(* CODESYS project plc_207_climat.project

Project tree, tasks and I/O mapping:
  Device : Owen SPK2xx 03.CS.WEB, Owen, order no. 023, version 3.5.4.20
    application Application
      libraries: Standard, * (System); VisuDialogs, * (System)
      task MainTask (cyclic, interval t#10ms, priority 1) calls PLC_PRG
      task VISU_TASK (cyclic, interval 100 ms, priority 31) calls VisuElems.Visu_Prg
      task AlarmManagerTask (cyclic, interval 50 ms, priority 31) calls AlarmManager.Alarm_Prg
      task Taskbus (cyclic, interval t#200ms, priority 1) calls MV110_16DN, MV110_8A, MU110_8P
      program PLC_PRG [ST]
      visualisation log_visu
      function two_word_to_real [ST]
      image pool ImagePool
      Alarm Configuration
        text list AlarmGroup
        alarm group AlarmGroup
            11 [Info]: Comparison Equal, ExpressionToCompare FALSE, Expression PLC_PRG.heating_on_level_1 - "Обогрев выключен, уровень 1"
            14 [Info]: Comparison Equal, ExpressionToCompare FALSE, Expression PLC_PRG.fire_alarm - "Пожара нет"
            8 [Info]: Comparison Equal, ExpressionToCompare FALSE, Expression PLC_PRG.air_valves_open - "Заслонки закрыты"
            9 [Info]: Comparison Equal, ExpressionToCompare FALSE, Expression PLC_PRG.fan_on_1 - "Вентилятор 1 выключен"
            12 [Info]: Comparison Equal, ExpressionToCompare FALSE, Expression PLC_PRG.heating_on_level_2 - "Обогрев выключен, уровень 2"
            0 [Error]: Comparison Equal, ExpressionToCompare TRUE, Expression PLC_PRG.air_valves_open - "Заслонки открыты"
            1 [Error]: Comparison Equal, ExpressionToCompare TRUE, Expression PLC_PRG.fan_on_1 - "Вентилятор 1 включен"
            2 [Error]: Comparison Equal, ExpressionToCompare TRUE, Expression PLC_PRG.fan_on_2 - "Вентилятор 2 включен"
            15 [Info]: Comparison Equal, ExpressionToCompare FALSE, Expression PLC_PRG.extinction_voltage - "Наличие напряжения на СШ"
            4 [Error]: Comparison Equal, ExpressionToCompare TRUE, Expression PLC_PRG.heating_on_level_2 - "Обогрев включен, уровень 2"
            5 [Error]: Comparison Equal, ExpressionToCompare TRUE, Expression PLC_PRG.automation_off - "Автоматика выключена"
            6 [Error]: Comparison Equal, ExpressionToCompare TRUE, Expression PLC_PRG.fire_alarm - "Пожар"
            7 [Error]: Comparison Equal, ExpressionToCompare TRUE, Expression PLC_PRG.extinction_voltage - "Исчезновение напряжения на СШ"
            13 [Info]: Comparison Equal, ExpressionToCompare TRUE, Expression PLC_PRG.automation_on - "Автоматика включена"
            3 [Error]: Comparison Equal, ExpressionToCompare TRUE, Expression PLC_PRG.heating_on_level_1 - "Обогрев включен, уровень 1"
            10 [Info]: Comparison Equal, ExpressionToCompare FALSE, Expression PLC_PRG.fan_on_2 - "Вентилятор 2 выключен"
        AlarmStorage
        alarm class Info (priority 10, acknowledge REP)
        alarm class Error (priority 20, acknowledge REP)
      visualisation log_visu_history
      function block BLINK [ST]
      visualisation main
      data type MAIN_STATE
    Modbus : Modbus COM, 3S - Smart Software Solutions GmbH, version 3.4.0.0
        settings: DataBits = 8; StopBits = 1; ComPort = 3
      Modbus_Master : Modbus Master, COM Port, 3S - Smart Software Solutions GmbH, version 3.5.4.0
          settings: Transmission = 'RTU'; ResponseTimeout = 300; TimeBetweenFrames = 50
        MV110_16DN : Modbus Slave, COM Port, 3S - Smart Software Solutions GmbH, version 3.5.4.0
            settings: SlaveAddress = 1; ResponseTimeout = 200; UseExtendedFunctionCodes = TRUE; Channel0.Function Code = 3; Channel0.Read Offset = 16#0033; Channel0.Read Length = 1; Channel0.Write Offset = 0; Channel0.Write Length = 0; Channel0.Cycle Time = 100
            input  Application.PLC_PRG.fan_on_1 : BOOL  // Channel0.Channel0.Bit0
            input  Application.PLC_PRG.fan_on_2 : BOOL  // Channel0.Channel0.Bit1
            input  Application.PLC_PRG.heating_on_level_1 : BOOL  // Channel0.Channel0.Bit2
            input  Application.PLC_PRG.heating_on_level_2 : BOOL  // Channel0.Channel0.Bit3
            input  Application.PLC_PRG.air_valves_open : BOOL  // Channel0.Channel0.Bit4
            input  Application.PLC_PRG.automation_off : BOOL  // Channel0.Channel0.Bit6
            input  Application.PLC_PRG.fire_alarm : BOOL  // Channel0.Channel0.Bit7
            input  Application.PLC_PRG.extinction_voltage_r : BOOL  // Channel0.Channel0.Bit8
            unmapped channels: Channel0
        MU110_8P : Modbus Slave, COM Port, 3S - Smart Software Solutions GmbH, version 3.5.4.0
            settings: SlaveAddress = 2; ResponseTimeout = 200; UseExtendedFunctionCodes = TRUE; Channel0.Function Code = 15; Channel0.Read Offset = 0; Channel0.Read Length = 0; Channel0.Write Offset = 16#0000; Channel0.Write Length = 8; Channel0.Cycle Time = 100
            output Application.PLC_PRG.ctr_vent : BOOL  // Channel0.Channel0.Bit0
            output Application.PLC_PRG.ctr_heating_level_1 : BOOL  // Channel0.Channel0.Bit1
            output Application.PLC_PRG.ctr_heating_level_2 : BOOL  // Channel0.Channel0.Bit2
            output Application.PLC_PRG.ctr_air_valves_open : BOOL  // Channel0.Channel0.Bit3
            output Application.PLC_PRG.ctr_low_temp_alarm : BOOL  // Channel0.Channel0.Bit4
            output Application.PLC_PRG.ctr_high_temp_alarm : BOOL  // Channel0.Channel0.Bit5
            output Application.PLC_PRG.ctr_fire_alarm : BOOL  // Channel0.Channel0.Bit6
            output Application.PLC_PRG.ctr_no_voltage_alarm : BOOL  // Channel0.Channel0.Bit7
            unmapped channels: Channel0
        MV110_8A : Modbus Slave, COM Port, 3S - Smart Software Solutions GmbH, version 3.5.4.0
            settings: SlaveAddress = 3; ResponseTimeout = 200; UseExtendedFunctionCodes = TRUE; Channel0.Function Code = 3; Channel0.Read Offset = 16#0004; Channel0.Read Length = 26; Channel0.Write Offset = 0; Channel0.Write Length = 0; Channel0.Cycle Time = 100
            input  Application.PLC_PRG.arr_t_outside[0] : WORD  // Channel0.Channel0
            input  Application.PLC_PRG.arr_t_outside[1] : WORD  // Channel0.Channel0
            input  Application.PLC_PRG.arr_t_inside_1[0] : WORD  // Channel0.Channel0
            input  Application.PLC_PRG.arr_t_inside_1[1] : WORD  // Channel0.Channel0
            input  Application.PLC_PRG.arr_t_inside_2[0] : WORD  // Channel0.Channel0
            input  Application.PLC_PRG.arr_t_inside_2[1] : WORD  // Channel0.Channel0
            unmapped channels: Channel0
    Modbus_OUT : Modbus COM, 3S - Smart Software Solutions GmbH, version 3.4.0.0
        settings: DataBits = 8; StopBits = 1; ComPort = 4
      Modbus_Slave : Modbus Serial Device, 3S - Smart Software Solutions GmbH, version 3.5.3.80
          settings: Unit-ID = 3
          output Application.PLC_PRG.fan_on_1 : BOOL  // Outputs.Outputs.Bit0
          output Application.PLC_PRG.fan_on_2 : BOOL  // Outputs.Outputs.Bit1
          output Application.PLC_PRG.heating_on_level_1 : BOOL  // Outputs.Outputs.Bit2
          output Application.PLC_PRG.heating_on_level_2 : BOOL  // Outputs.Outputs.Bit3
          output Application.PLC_PRG.air_valves_open : BOOL  // Outputs.Outputs.Bit4
          output Application.PLC_PRG.automation_off : BOOL  // Outputs.Outputs.Bit5
          output Application.PLC_PRG.fire_alarm : BOOL  // Outputs.Outputs.Bit6
          output Application.PLC_PRG.extinction_voltage_r : BOOL  // Outputs.Outputs.Bit7
          output Application.PLC_PRG.ctr_low_temp_alarm : BOOL  // Outputs.Outputs.Bit8
          output Application.PLC_PRG.ctr_high_temp_alarm : BOOL  // Outputs.Outputs.Bit9
          output Application.PLC_PRG.arr_t_outside[0] : WORD  // Outputs.Outputs
          output Application.PLC_PRG.arr_t_outside[1] : WORD  // Outputs.Outputs
          output Application.PLC_PRG.arr_t_inside_1[0] : WORD  // Outputs.Outputs
          output Application.PLC_PRG.arr_t_inside_1[1] : WORD  // Outputs.Outputs
          output Application.PLC_PRG.arr_t_inside_2[0] : WORD  // Outputs.Outputs
          output Application.PLC_PRG.arr_t_inside_2[1] : WORD  // Outputs.Outputs
          unmapped channels: Inputs, Outputs
  text list GlobalTextList
  5ce3da45-db07-42e7-a21c-a00fff4ed8f6|D:\по щсу\ДЭС\visu\zit.jpg
  5ce3da45-db07-42e7-a21c-a00fff4ed8f6|D:\по щсу\ДЭС\visu\entel.jpg
  5ce3da45-db07-42e7-a21c-a00fff4ed8f6|C:\Users\Maxim\Desktop\mie110-3m.jpg
  5ce3da45-db07-42e7-a21c-a00fff4ed8f6|C:\Users\Maxim\Desktop\warning2.jpg
  global variables GVL
  5ce3da45-db07-42e7-a21c-a00fff4ed8f6|C:\Users\Maxim\Desktop\SHM96.png
*)

// Device/Application/MAIN_STATE
TYPE MAIN_STATE :
(
	IDLE,
	HEATING_LEVEL_ONE,
	HEATING_LEVEL_TWO,
	FANS
);
END_TYPE

// GVL
VAR_GLOBAL PERSISTENT RETAIN
	login:STRING:='U';
	pass:STRING:='13';
	zavod_number:STRING;
	datta:STRING;
END_VAR

// Device/Application/PLC_PRG
PROGRAM PLC_PRG
VAR	

current_state		: MAIN_STATE := IDLE;
//------------- Состояние коненого автомата работы климата -------------//
temp_min_alarm		: REAL := 8;
temp_hight_alarm	: REAL := 30;

temp_heating_one_on	: REAL := 10; // Температура включения обогрева, уровень 1
temp_heating_two_on	: REAL := 8; // Температура включения обогрева, уровень 2
temp_heating_off	: REAL := 18; // Температура выключения обогрева

temp_air_valves_on	: REAL := 12; // Минимальная температура открытых заслонок
temp_air_valves_off	: REAL := 10; // Температура закрытия заслонок
temp_air_valves		: REAL := temp_air_valves_on; // Минимальная температура открытых заслонок

temp_fans_on		: REAL := 23; // Температура включения вентиляторов
temp_fans_off		: REAL := 18; // Температура выключения вентиляторов
temp_max_outdoor	: REAL := 25; // Не включать вентиляторы при уличной температуре больше этого значения 

//-------------------------------- Состояния --------------------------------//
fan_on_1 			: BOOL;
fan_on_2 			: BOOL;
heating_on_level_1 	: BOOL;
heating_on_level_2 	: BOOL;
air_valves_open 	: BOOL;
automation_off		: BOOL;
fire_alarm 			: BOOL;
extinction_voltage_r: BOOL;	// инверсия

extinction_voltage	: BOOL;
automation_on		: BOOL;
//-------------------------------- Состояния --------------------------------//

//-------------------------- Температурные датчики --------------------------//
//входные аналоговые сигналы с температурных датчиков
arr_t_outside		: ARRAY[0..1] OF WORD;
arr_t_inside_1		: ARRAY[0..1] OF WORD;
arr_t_inside_2		: ARRAY[0..1] OF WORD;
pT_inside 			: POINTER TO ARRAY [0..1] OF WORD;
pT_outside			: POINTER TO ARRAY [0..1] OF WORD;

temp_outside		: REAL; // значение с датчика уличной температуры
temp_inside			: REAL; // значение внутренней температуры
temp_inside_1		: REAL; // значение с 1ого внутренного датчика температуры
temp_inside_2		: REAL; // значение со 2ого внутреннего датчика температуры
//-------------------------- Температурные датчики --------------------------//

//----------------- Управляющие выходные сигналы на блок МУ -----------------//
ctr_vent			:BOOL; // перерменная подачи команды на вентиляторы
ctr_heating_level_1	:BOOL; // перерменная подачи команды на обогрев, уровень 1
ctr_heating_level_2	:BOOL; // перерменная подачи команды на обогрев, уровень 2
ctr_air_valves_open	:BOOL; // переменная подачи команды на воздушные клапаны
ctr_low_temp_alarm	:BOOL; // тревога для телемеханики "Низкая температура"
ctr_high_temp_alarm	:BOOL; // тревога для телемеханики "Высокая температура"
ctr_fire_alarm		:BOOL; // тревога для телемеханики "Пожар"
ctr_no_voltage_alarm:BOOL; // тревога для телемеханики "Нет напряжения на СШ"
//----------------- Управляющие выходные сигналы на блок МУ -----------------//

//------------------ Перезапуск подключения по Modbus ------------------//
blink_time  		: TIME := T#150MS;
blink_16DN			: BLINK;
blink_8A			: BLINK;
blink_8P			: BLINK;
//------------------ Перезапуск подключения по Modbus ------------------//

main_delay			: TON; // Задержка запуска основной функции
main_delay_time		: TIME := T#5S;

visu_true			: BOOL := TRUE;
END_VAR

automation_on := NOT(automation_off);
extinction_voltage := NOT(extinction_voltage_r);

//------------------ Перезапуск подключения по Modbus ------------------//
IF MV110_16DN.xError THEN
	blink_16DN(ENABLE := TRUE, TIMELOW := blink_time, TIMEHIGH := blink_time);
	MV110_16DN.xReset := blink_16DN.OUT;
END_IF

IF MU110_8P.xError THEN	
	blink_8P(ENABLE := TRUE, TIMELOW := blink_time, TIMEHIGH := blink_time);
	MU110_8P.xReset := blink_8P.OUT;
END_IF

IF MV110_8A.xError THEN	
	blink_8A(ENABLE := TRUE, TIMELOW := blink_time, TIMEHIGH := blink_time);
	MV110_8A.xReset := blink_8A.OUT;
END_IF
//------------------ Перезапуск подключения по Modbus ------------------//

// преобразование получаемых переменных от МВ110_8А типа WORD  в Real
pT_outside := ADR(arr_t_outside);
temp_outside := two_word_to_real(pT_outside);

pT_inside := ADR(arr_t_inside_1);
temp_inside_1 := two_word_to_real(pT_inside);
pT_inside := ADR(arr_t_inside_2);
temp_inside_2 := two_word_to_real(pT_inside);
temp_inside := (temp_inside_1 + temp_inside_2) / 2;

main_delay(IN := TRUE, PT := main_delay_time);
IF main_delay.Q=1 THEN
	// Установка тревоги для телемеханики "Нет напряжения на СШ"
	ctr_no_voltage_alarm := extinction_voltage;
	
	//** Определение высокой и низкой температур **/
	IF temp_inside < temp_min_alarm THEN
		ctr_low_temp_alarm := TRUE;
	ELSE
		ctr_low_temp_alarm := FALSE;
	END_IF
	
	IF temp_inside > temp_hight_alarm THEN
		ctr_high_temp_alarm := TRUE;
	ELSE
		ctr_high_temp_alarm := FALSE;
	END_IF
	//** Определение высокой и низкой температур **/
	
	IF temp_outside > temp_air_valves THEN			//** Открытие заслонок **//
		ctr_air_valves_open := TRUE;
		temp_air_valves := temp_air_valves_off;
	ELSE
		ctr_air_valves_open := FALSE;
		temp_air_valves := temp_air_valves_on;
	END_IF
	
	IF fire_alarm = TRUE THEN						//** Пожар **//
		ctr_heating_level_1 := FALSE;
		ctr_heating_level_2	:= FALSE;
		ctr_vent := FALSE;
		ctr_air_valves_open := FALSE;
		ctr_fire_alarm := TRUE;
	ELSIF automation_off = FALSE THEN				//** Нормальный режим работы **//
		CASE current_state OF
		IDLE:											//** Режим простоя **//
			ctr_heating_level_1 := FALSE;
			ctr_heating_level_2	:= FALSE;
			ctr_vent := FALSE;
			ctr_fire_alarm := FALSE;
			
			IF temp_inside >= temp_fans_on AND  temp_outside <= temp_max_outdoor THEN
				current_state := FANS;
			ELSIF temp_inside <= temp_heating_one_on THEN
				current_state := HEATING_LEVEL_ONE;
			END_IF
		HEATING_LEVEL_ONE:										//** Режим обогрева, уровень 1 **//
			ctr_heating_level_1 := TRUE;
			ctr_heating_level_2	:= FALSE;
			ctr_vent := FALSE;
			ctr_fire_alarm := FALSE;
			
			IF temp_inside >= temp_heating_off THEN
				current_state := IDLE;
			ELSIF temp_inside <= temp_heating_two_on THEN
				current_state := HEATING_LEVEL_TWO;
			END_IF
		HEATING_LEVEL_TWO:										//** Режим обогрева, уровень 2 **//
			ctr_vent := FALSE;
			ctr_heating_level_1 := TRUE;
			ctr_heating_level_2	:= TRUE;
			ctr_fire_alarm := FALSE;
			
			IF temp_inside >= temp_heating_off THEN
				current_state := IDLE;
			END_IF
		FANS:													//** Режим вентиляции **//
			ctr_vent := TRUE;
			ctr_air_valves_open := TRUE;
			ctr_heating_level_1 := FALSE;
			ctr_heating_level_2	:= FALSE;
			ctr_fire_alarm := FALSE;
			
			IF temp_inside <= temp_fans_off OR temp_outside >= temp_max_outdoor THEN
				current_state := IDLE;
			END_IF
		END_CASE
	ELSE											//** Автоматика отключена **//
		ctr_vent := FALSE;
		ctr_heating_level_1 := FALSE;
		ctr_heating_level_2	:= FALSE;
		ctr_air_valves_open	:= FALSE;
		ctr_fire_alarm := FALSE;
	END_IF
END_IF

END_PROGRAM

// Device/Application/two_word_to_real
FUNCTION two_word_to_real : real
VAR_INPUT
	IN_Data: POINTER TO ARRAY[0..1] OF WORD; (*Указатель на массив регистров для Float*)
END_VAR

VAR
	p1: POINTER TO BYTE;
	p2: POINTER TO BYTE;
END_VAR

p1:=ADR(two_word_to_real);
p2:=ADR(IN_Data^[1]);
p1^:=p2^;
p1:=p1+1;
p2:=p2+1;
p1^:=p2^;
p1:=p1+1;
p2:=ADR(IN_Data^[0]);
p1^:=p2^;
p1:=p1+1;
p2:=p2+1;
p1^:=p2^;

END_FUNCTION

// Device/Application/BLINK

FUNCTION_BLOCK BLINK
(* Function block to simulate a turn signal *)
VAR_INPUT
	ENABLE:BOOL;		(* TRUE:run Blink, FALSE: OUT keeps its value*)
	TIMELOW:TIME;		(* Time for OUT=FALSE *)
	TIMEHIGH:TIME;		(* Time for OUT=TRUE *)
END_VAR
VAR_OUTPUT
	OUT:BOOL;			(* output variable, starting with FALSE *)
END_VAR
VAR
	CLOCK:TP;
END_VAR

CLOCK();										(* call Timer *)
IF CLOCK.Q=FALSE AND ENABLE THEN	(* time passed or init *)
	CLOCK(IN:=FALSE);						(* reset Timer *)
	CLOCK(IN:=TRUE);						(* restart Timer *)
	IF OUT=FALSE THEN
		CLOCK.PT:=TIMEHIGH;
	ELSE
		CLOCK.PT:=TIMELOW;
	END_IF;
							(* invert *)
END_IF
OUT := NOT out;

END_FUNCTION_BLOCK

// Device/Application/log_visu
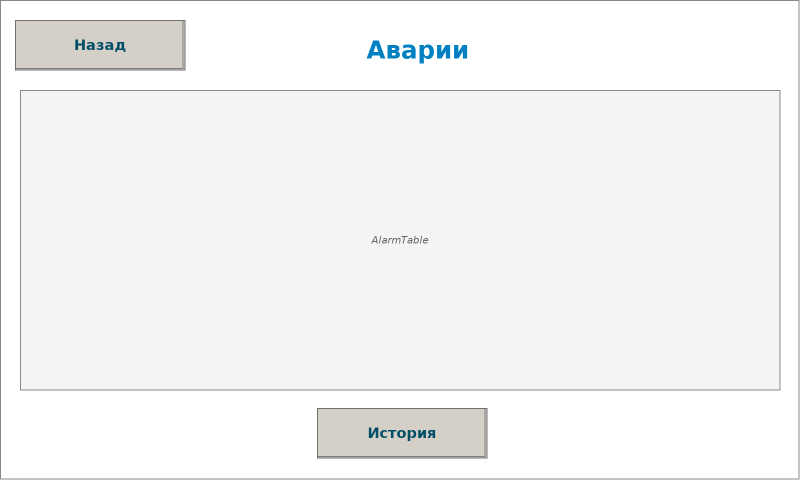
VISUALIZATION log_visu  // 800x480, background image ImagePool.bg_800
    Button (15,20 170x50), "Назад"
        OnMouseClick:  Assign=main, Type=Assignment
    AlarmTable (20,90 760x300)
        Column[0]: ColumnTitle=Временная отметка
        Column[1]: ColumnTitle=Сообщение
        p1521930926: AlarmGroup
        p1663851261: __All
    Rectangle (215,35 406x30), "Аварии"
    Button (317,408 170x50), "История"
        OnMouseClick:  Assign=log_visu_history, Type=Assignment
    hotkey  Id=481037385728, Key=KeyDown=True, KeyName=0, VisuElemId=6
    hotkey  Id=481038434304, Key=KeyName=0, VisuElemId=6
    hotkey  Id=481037385728, Key=KeyDown=True, KeyName=0, VisuElemId=17
    hotkey  Id=481038434304, Key=KeyName=0, VisuElemId=17
END_VISUALIZATION

// Device/Application/log_visu_history
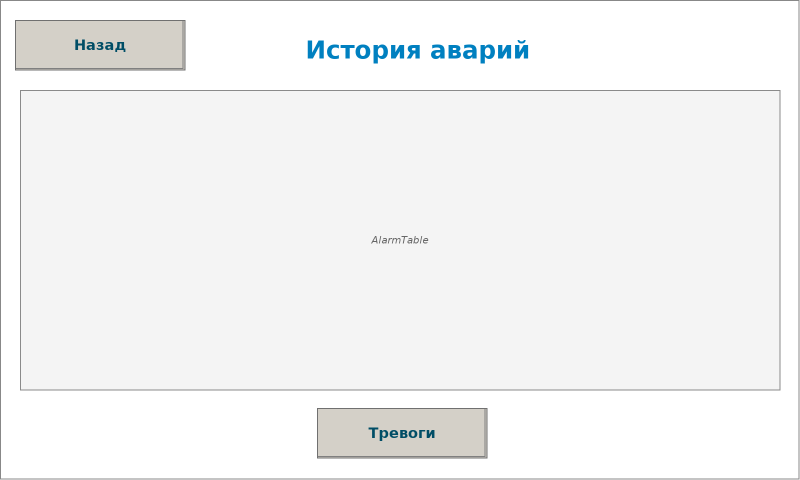
VISUALIZATION log_visu_history  // 800x480, background image ImagePool.bg_800
    Button (15,20 170x50), "Назад"
        OnMouseClick:  Assign=main, Type=Assignment
    AlarmTable (20,90 760x300)
        Column[0]: ColumnTitle=Временная отметка
        Column[1]: ColumnTitle=Сообщение
        p1521930926: AlarmGroup
        p1663851261: __All
        p3266827225: PLC_PRG.visu_true
    Rectangle (215,35 406x30), "История аварий"
    Button (317,408 170x50), "Тревоги"
        OnMouseClick:  Assign=log_visu, Type=Assignment
    hotkey  Id=481037385728, Key=KeyDown=True, KeyName=0, VisuElemId=6
    hotkey  Id=481038434304, Key=KeyName=0, VisuElemId=6
    hotkey  Id=481037385728, Key=KeyDown=True, KeyName=0, VisuElemId=17
    hotkey  Id=481038434304, Key=KeyName=0, VisuElemId=17
END_VISUALIZATION

// Device/Application/main
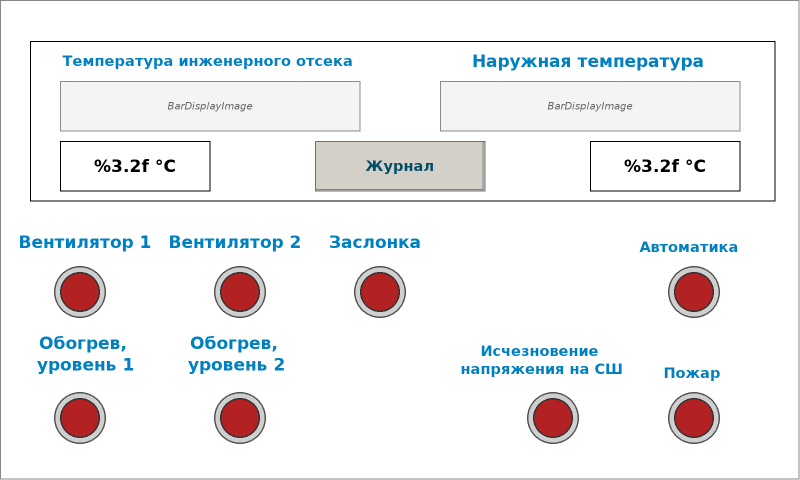
VISUALIZATION main  // 800x480, background image ImagePool.bg_800
    Rectangle (30,41 745x160)
    Rectangle (35,46 346x30), "Температура инженерного отсека"
    Rectangle (60,141 150x50), "%3.2f °С", text variable: PLC_PRG.temp_inside
    BarDisplayImage (60,81 300x50), value: PLC_PRG.temp_inside, style: BarDisplayImage-Gray, scale format: %.1f, scale -10..50
    Rectangle (415,46 346x30), "Наружная температура"
    Rectangle (590,141 150x50), "%3.2f °С", text variable: PLC_PRG.temp_outside
    BarDisplayImage (440,81 300x50), value: PLC_PRG.temp_outside, style: BarDisplayImage-Gray, scale format: %.1f, scale -60..80
    Rectangle (614,232 150x30), "Автоматика"
    Lamp1 (664,262 60x60), variable: PLC_PRG.automation_on, style: Lamp-Lamp1-Red
    Lamp1 (50,262 60x60), variable: PLC_PRG.fan_on_1, style: Lamp-Lamp1-Red
    Rectangle (10,232 150x20), "Вентилятор 1"
    Lamp1 (350,262 60x60), variable: PLC_PRG.air_valves_open, style: Lamp-Lamp1-Red
    Rectangle (320,232 110x20), "Заслонка"
    Lamp1 (210,388 60x60), variable: PLC_PRG.heating_on_level_2, style: Lamp-Lamp1-Red
    Lamp1 (210,262 60x60), variable: PLC_PRG.fan_on_2, style: Lamp-Lamp1-Red
    Rectangle (160,232 150x20), "Вентилятор 2"
    Button (315,141 170x50), "Журнал"
        OnMouseClick:  Assign=log_visu, Type=Assignment
    Lamp1 (50,388 60x60), variable: PLC_PRG.heating_on_level_1, style: Lamp-Lamp1-Red
    Rectangle (8,331 150x46), "Обогрев, уровень 1"
    Rectangle (159,331 150x46), "Обогрев, уровень 2"
    Rectangle (617,358 150x30), "Пожар"
    Lamp1 (664,388 60x60), variable: PLC_PRG.fire_alarm, style: Lamp-Lamp1-Red
    Rectangle (434,341 216x38), "Исчезновение напряжения на СШ"
    Lamp1 (523,388 60x60), variable: PLC_PRG.extinction_voltage, style: Lamp-Lamp1-Red
END_VISUALIZATION

(* text list AlarmGroup (id | default)
  8 | Заслонки закрыты
  9 | Вентилятор 1 выключен
  10 | Вентилятор 2 выключен
  11 | Обогрев выключен, уровень 1
  12 | Обогрев выключен, уровень 2
  13 | Автоматика включена
  14 | Пожара нет
  15 | Наличие напряжения на СШ
  7 | Исчезновение напряжения на СШ
  6 | Пожар
  5 | Автоматика выключена
  4 | Обогрев включен, уровень 2
  3 | Обогрев включен, уровень 1
  2 | Вентилятор 2 включен
  1 | Вентилятор 1 включен
  0 | Заслонки открыты
   |  *)
